FUNCTION_BLOCK FB_TcLogger IMPLEMENTS I_Logger
VAR_INPUT
END_VAR
VAR_OUTPUT
END_VAR
VAR_IN_OUT

END_VAR
VAR
END_VAR

METHOD M_Log
VAR_INPUT
	stEvent	: 		ST_Event;
END_VAR
IF stEvent.New THEN
	CASE stEvent.EventType OF
		E_Event.Error:
			ADSLOGSTR( msgCtrlMask := ADSLOG_MSGTYPE_ERROR , msgFmtStr := stEvent.Message, strArg := '');
		E_Event.Warning:
			ADSLOGSTR( msgCtrlMask := ADSLOG_MSGTYPE_WARN , msgFmtStr := stEvent.Message, strArg := '');
		E_Event.Information:
			ADSLOGSTR( msgCtrlMask := ADSLOG_MSGTYPE_HINT , msgFmtStr := stEvent.Message, strArg := '');
		E_Event.Debug:
			ADSLOGSTR( msgCtrlMask := ADSLOG_MSGTYPE_HINT, msgFmtStr := stEvent.Message, strArg := '');
		E_Event.Verbose:
			ADSLOGSTR( msgCtrlMask := ADSLOG_MSGTYPE_HINT , msgFmtStr := stEvent.Message, strArg := '');
	END_CASE
END_IF
END_METHOD

END_FUNCTION_BLOCK

(* stored: Version 1.1.0.1, ProductVersion 3.1.4024.12
   POU FB_TcLogger: Id {0039f59e-4c40-42a4-8ff2-37da92726d34}, SpecialFunc None
   Method M_Log: Id {8cf2d68c-783c-4dc8-a302-c8f0b2e2f3c8} *)
